(*
SPDX-FileCopyrightText: © 2026 Oleksandr Tiutyk <trofimich@gmail.com>
SPDX-License-Identifier: MIT
License: https://opensource.org/license/mit
*)

FUNCTION_BLOCK RandomTest EXTENDS TcUnit.FB_TestSuite
VAR
	{attribute 'hide'} 
	_ClassName : STRING := __POUNAME();	
END_VAR

GetInRange();
GetWithDispersion();
GetWithDispersionPercent();

{attribute 'monitoring' := 'call'}
PROPERTY ClassName : REFERENCE TO STRING
GET
ClassName REF= _ClassName;
END_GET
END_PROPERTY

METHOD GetInRange
VAR
	i : INT;
	
	value : LREAL;
END_VAR
VAR_INST
	testFinished : BOOL;
END_VAR
IF testFinished THEN 
	RETURN; 
END_IF 

TEST(__POUNAME());

FOR i := 0 TO 20 DO
	value := TOF_Core.Random.GetInRange(100, 200);
	
	IF value < 100 OR_ELSE value > 200 THEN
		AssertEquals_BOOL(TRUE, FALSE, 'Invalid GetInRange() implementation');
		RETURN;
	END_IF
END_FOR

testFinished := TRUE; 
TEST_FINISHED();
END_METHOD

METHOD GetWithDispersion
VAR
	i : INT;
	
	value : LREAL;
END_VAR
VAR_INST
	testFinished : BOOL;
END_VAR
IF testFinished THEN 
	RETURN; 
END_IF 

TEST(__POUNAME());

FOR i := 0 TO 20 DO
	value := TOF_Core.Random.GetWithDispersion(100, 10);
	
	IF value < 90 OR_ELSE value > 110 THEN
		AssertEquals_BOOL(TRUE, FALSE, 'Invalid GetWithDispersion() implementation');
		RETURN;
	END_IF
END_FOR

testFinished := TRUE; 

TEST_FINISHED();
END_METHOD

METHOD GetWithDispersionPercent
VAR
	i : INT;
	
	value : LREAL;
END_VAR
VAR_INST
	testFinished : BOOL;
END_VAR
IF testFinished THEN 
	RETURN; 
END_IF 

TEST(__POUNAME());


FOR i := 0 TO 20 DO
	value := TOF_Core.Random.GetWithDispersionPercent(100, 10);
	
	IF value < 90 OR_ELSE value > 110 THEN
		AssertEquals_BOOL(TRUE, FALSE, 'Invalid GetWithDispersionPercent() implementation');
		RETURN;
	END_IF
END_FOR

testFinished := TRUE; 
TEST_FINISHED();
END_METHOD

{attribute 'monitoring' := 'call'}
PROPERTY NamespaceName : REFERENCE TO STRING
GET
NamespaceName REF= CurrentNamespace.Name;
END_GET
END_PROPERTY

END_FUNCTION_BLOCK

(* stored: Version 1.1.0.1, ProductVersion 3.1.4026.20
   POU RandomTest: Id {2bc575a5-a2e8-41d3-a88b-91900261e812}, SpecialFunc None
   Property ClassName: Id {c63098eb-f1d1-4659-8651-4218958d4856}
   Get Get: Id {f3462718-1a95-4c40-b661-2789caf059a3}
   Method GetInRange: Id {9bc3a55f-15d0-4425-9ace-c713fc938781}
   Method GetWithDispersion: Id {4394b0e8-9382-436f-8ceb-d1938e9dcfdf}
   Method GetWithDispersionPercent: Id {5c23b097-6f9c-4d39-83e0-30e50ffd0a75}
   Property NamespaceName: Id {ed1a6086-9f9b-4d07-80f4-26fbd096eecc}
   Get Get: Id {2ce69c62-77bc-4051-99dc-71c5c5eadfd4} *)
